// TIA Portal V21 export
ORGANIZATION_BLOCK "Main"   // OB1, LAD, ProgramCycle
TITLE = "Main Program Sweep (Cycle)"
{ S7_Optimized_Access := 'TRUE' }
// stored: SetENOAutomatically false
BEGIN

REGION Network 2 (SCL)
   "Data_block_1"."zmienna 1" := "Data_block_1"."zmienna 2";
END_REGION
END_ORGANIZATION_BLOCK
